INTERFACE I_TargetZSensor

PROPERTY P_bSensor : BOOL
GET
END_GET
END_PROPERTY

END_INTERFACE

(* stored: Version 1.1.0.1, ProductVersion 3.1.0.25
   Itf I_TargetZSensor: Id {e54d7a9f-6c6f-442d-bb20-3947619f046d}
   Property P_bSensor: Id {ffb74354-aa81-4afc-9d2b-30544494b891}
   Get Get: Id {4cfe8a2f-d218-443c-84b3-81e0c1761036} *)
